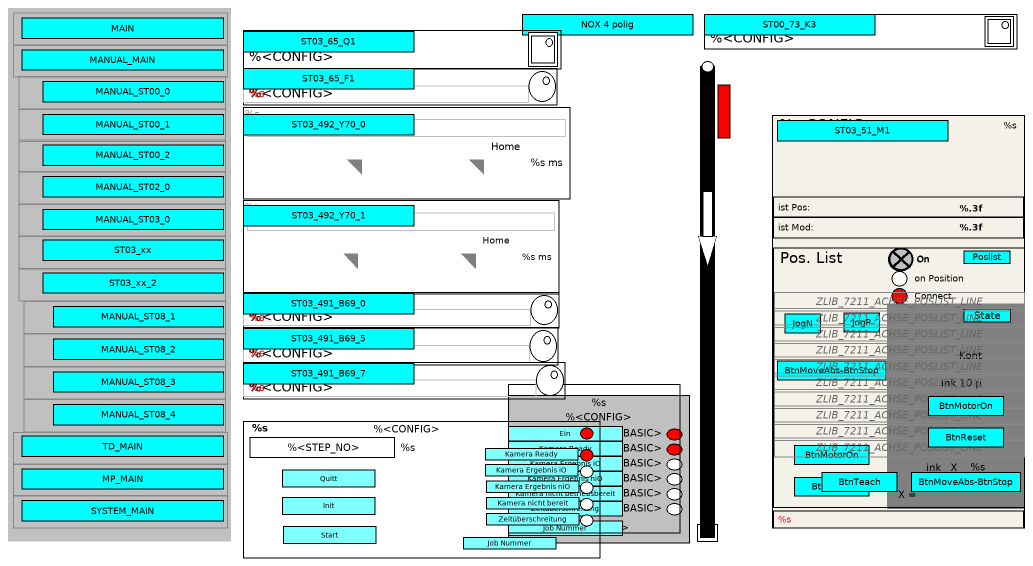
[picture p109: MANUAL_ST03_11 (HMI screen)]
embedded screen at (3,115)-(226,648): M0000_Manual
embedded screen at (238,214)-(565,306): ZLIB_VALVE_1_SENSORS
embedded screen at (238,307)-(554,401): ZLIB_VALVE_1_SENSORS
embedded screen at (238,399)-(554,435): VDIGIN
embedded screen at (238,434)-(553,472): VDIGIN
embedded screen at (767,222)-(1021,635): ZLIB_7211_Achse
embedded screen at (503,168)-(725,650): ZUFUEHRUNG_NOX_4POL
rectangle at (517,121)-(688,142): text "NOX 4 polig"; invisible if TRUE
rectangle at (238,312)-(409,333): text "ST03_492_Y70_1"; invisible if TRUE
rectangle at (238,221)-(409,242): text "ST03_492_Y70_0"; invisible if TRUE
rectangle at (238,400)-(409,421): text "ST03_491_B69_0"; invisible if TRUE
rectangle at (238,435)-(409,456): text "ST03_491_B69_5"; invisible if TRUE
rectangle at (772,227)-(943,248): text "ST03_51_M1"; invisible if TRUE
embedded screen at (238,137)-(556,176): VDIGOUT_SMAL
rectangle at (238,138)-(409,159): text "ST03_65_Q1"; invisible if TRUE
embedded screen at (238,175)-(552,212): VDIGIN
rectangle at (238,175)-(409,196): text "ST03_65_F1"; invisible if TRUE
embedded screen at (699,121)-(1012,156): VDIGOUT_SMAL
rectangle at (699,121)-(870,142): text "ST00_73_K3"; invisible if TRUE
embedded screen at (238,528)-(595,665): ZLIB_SENSOPART_4
embedded screen at (238,469)-(560,506): VDIGIN
rectangle at (238,470)-(409,491): text "ST03_491_B69_7"; invisible if TRUE
1 more shapes without text or variables
*)

(* Visualisation 01_ManualMode/ST03/MANUAL_ST03_12
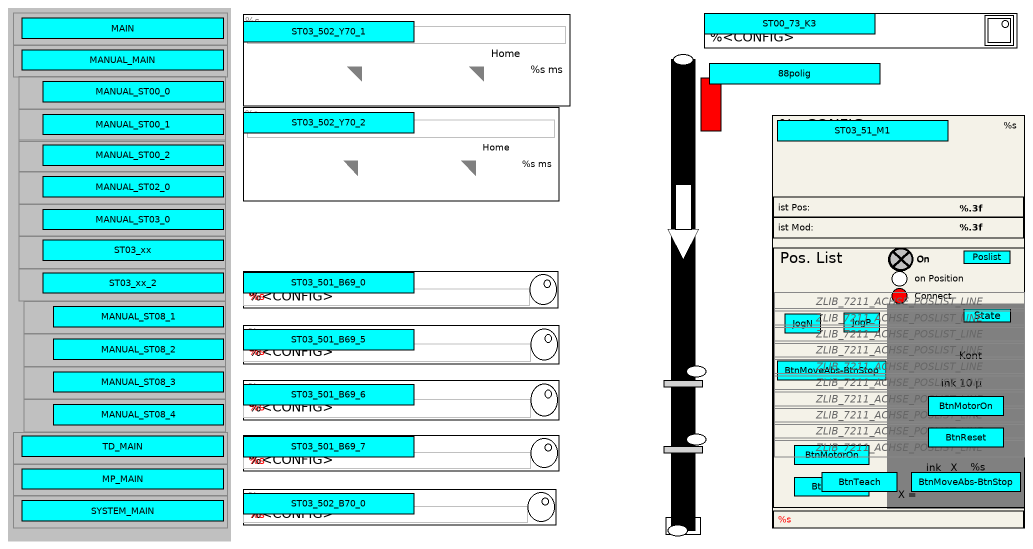
embedded screen at (3,115)-(226,648): M0000_Manual
embedded screen at (238,121)-(565,213): ZLIB_VALVE_1_SENSORS
embedded screen at (238,214)-(554,308): ZLIB_VALVE_1_SENSORS
embedded screen at (238,542)-(554,578): VDIGIN
embedded screen at (238,596)-(551,632): VDIGIN
embedded screen at (767,222)-(1021,635): ZLIB_7211_Achse
embedded screen at (646,161)-(716,643): ZUFUEHRUNG_88POL
rectangle at (704,170)-(875,191): text "88polig"; invisible if TRUE
rectangle at (238,219)-(409,240): text "ST03_502_Y70_2"; invisible if TRUE
rectangle at (238,128)-(409,149): text "ST03_502_Y70_1"; invisible if TRUE
rectangle at (238,543)-(409,564): text "ST03_501_B69_7"; invisible if TRUE
rectangle at (238,600)-(409,621): text "ST03_502_B70_0"; invisible if TRUE
rectangle at (772,227)-(943,248): text "ST03_51_M1"; invisible if TRUE
embedded screen at (238,487)-(554,527): VDIGIN
embedded screen at (238,378)-(553,415): VDIGIN
embedded screen at (238,432)-(554,471): VDIGIN
rectangle at (238,379)-(409,400): text "ST03_501_B69_0"; invisible if TRUE
rectangle at (238,436)-(409,457): text "ST03_501_B69_5"; invisible if TRUE
rectangle at (238,491)-(409,512): text "ST03_501_B69_6"; invisible if TRUE
embedded screen at (699,120)-(1012,155): VDIGOUT_SMAL
rectangle at (699,120)-(870,141): text "ST00_73_K3"; invisible if TRUE
*)

(* Visualisation 01_ManualMode/ST03/MANUAL_ST03_13
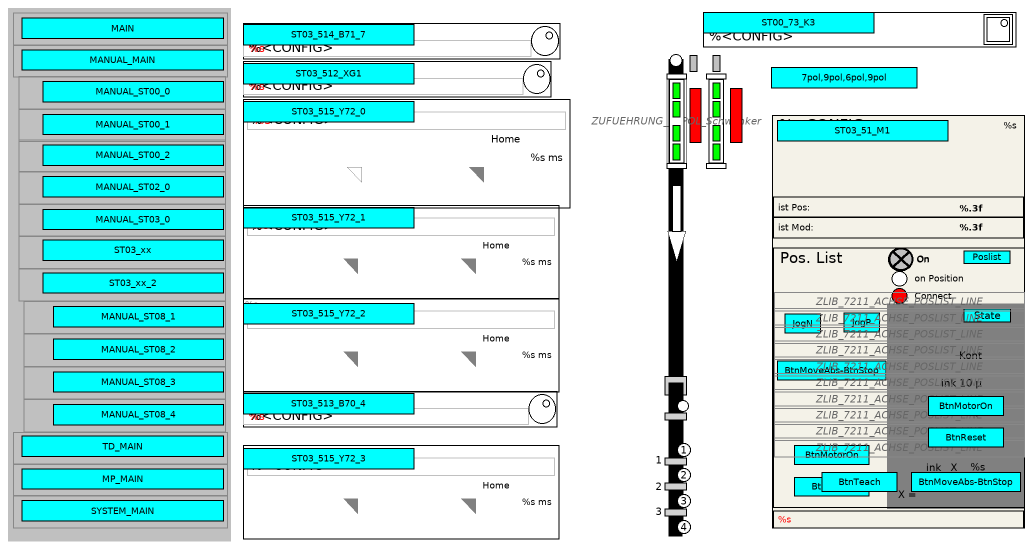
embedded screen at (3,115)-(226,648): M0000_Manual
embedded screen at (238,312)-(554,406): ZLIB_VALVE_1_SENSORS
embedded screen at (238,130)-(555,166): VDIGIN
embedded screen at (767,222)-(1021,635): ZLIB_7211_Achse
embedded screen at (646,161)-(737,643): ZUFUEHRUNG_7POL
rectangle at (766,174)-(912,195): text "7pol,9pol,6pol,9pol"; invisible if TRUE
rectangle at (238,314)-(409,335): text "ST03_515_Y72_1"; invisible if TRUE
rectangle at (238,131)-(409,152): text "ST03_514_B71_7"; invisible if TRUE
rectangle at (772,227)-(943,248): text "ST03_51_M1"; invisible if TRUE
embedded screen at (238,168)-(546,204): VDIGIN
rectangle at (238,170)-(409,191): text "ST03_512_XG1"; invisible if TRUE
embedded screen at (238,405)-(554,499): ZLIB_VALVE_1_SENSORS
embedded screen at (238,498)-(552,534): VDIGIN
rectangle at (238,410)-(409,431): text "ST03_515_Y72_2"; invisible if TRUE
rectangle at (238,500)-(409,521): text "ST03_513_B70_4"; invisible if TRUE
embedded screen at (238,552)-(554,646): ZLIB_VALVE_1_SENSORS
rectangle at (238,555)-(409,576): text "ST03_515_Y72_3"; invisible if TRUE
embedded screen at (238,206)-(565,315): ZLIB_VALVE_2_SENSORS
rectangle at (238,208)-(409,229): text "ST03_515_Y72_0"; invisible if TRUE
embedded screen at (698,119)-(1011,154): VDIGOUT_SMAL
rectangle at (698,119)-(869,140): text "ST00_73_K3"; invisible if TRUE
*)

(* Visualisation 01_ManualMode/ST03/MANUAL_ST03_13_2
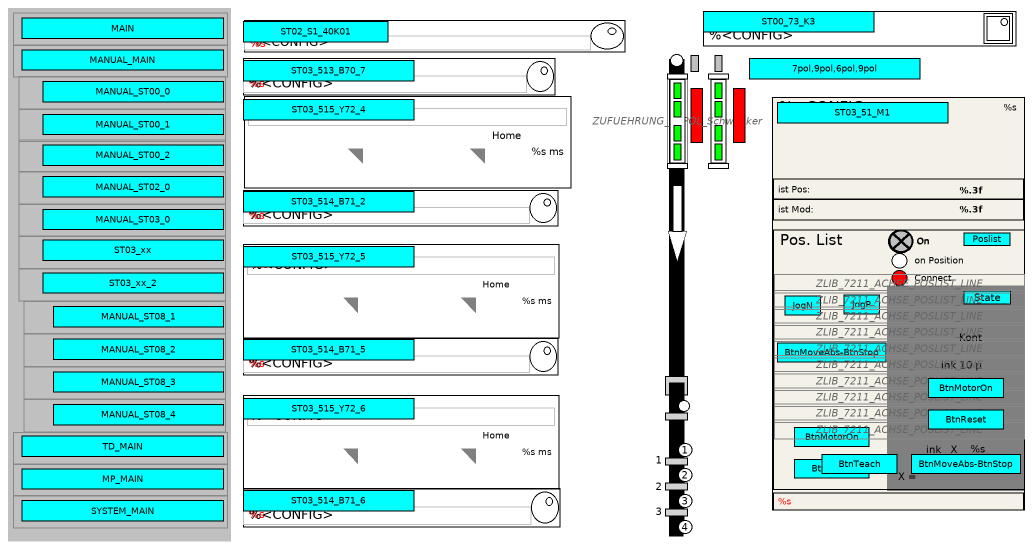
embedded screen at (3,115)-(226,648): M0000_Manual
embedded screen at (239,203)-(566,295): ZLIB_VALVE_1_SENSORS
embedded screen at (238,351)-(554,445): ZLIB_VALVE_1_SENSORS
embedded screen at (238,445)-(553,482): VDIGIN
embedded screen at (767,204)-(1021,617): ZLIB_7211_Achse
embedded screen at (646,161)-(740,643): ZUFUEHRUNG_7POL
rectangle at (744,165)-(915,186): text "7pol,9pol,6pol,9pol"; invisible if TRUE
rectangle at (238,353)-(409,374): text "ST03_515_Y72_5"; invisible if TRUE
rectangle at (238,206)-(409,227): text "ST03_515_Y72_4"; invisible if TRUE
rectangle at (238,446)-(409,467): text "ST03_514_B71_5"; invisible if TRUE
rectangle at (772,209)-(943,230): text "ST03_51_M1"; invisible if TRUE
embedded screen at (238,165)-(550,202): VDIGIN
rectangle at (238,167)-(409,188): text "ST03_513_B70_7"; invisible if TRUE
embedded screen at (238,502)-(554,596): ZLIB_VALVE_1_SENSORS
embedded screen at (238,595)-(555,634): VDIGIN
rectangle at (238,505)-(409,526): text "ST03_515_Y72_6"; invisible if TRUE
rectangle at (238,597)-(409,618): text "ST03_514_B71_6"; invisible if TRUE
embedded screen at (238,297)-(553,333): VDIGIN
rectangle at (238,298)-(409,319): text "ST03_514_B71_2"; invisible if TRUE
embedded screen at (239,127)-(620,159): VDIGIN
rectangle at (238,128)-(383,149): text "ST02_S1_40K01"; invisible if TRUE
embedded screen at (698,118)-(1011,153): VDIGOUT_SMAL
rectangle at (698,118)-(869,139): text "ST00_73_K3"; invisible if TRUE
*)

(* Visualisation 01_ManualMode/ST03/MANUAL_ST03_14
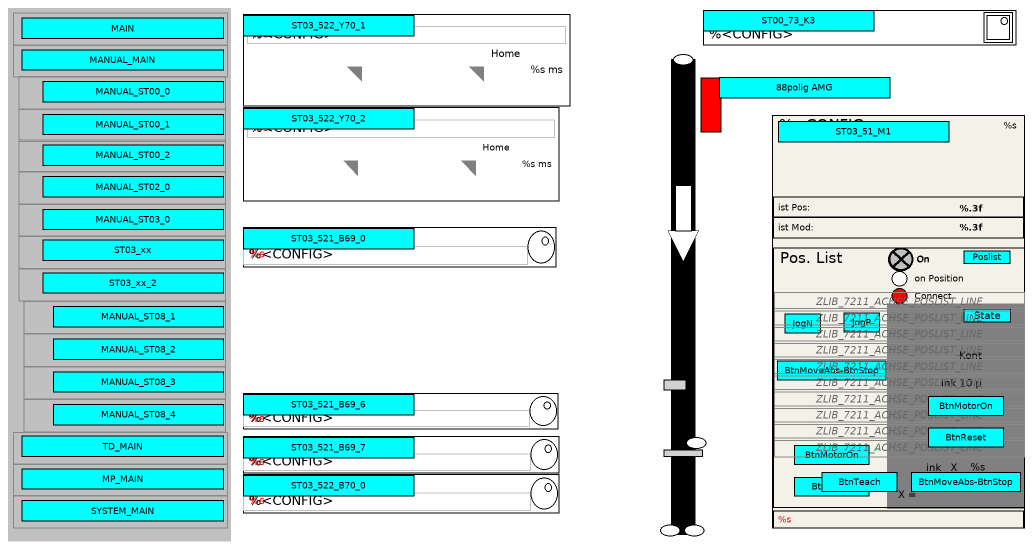
embedded screen at (3,115)-(226,648): M0000_Manual
embedded screen at (238,121)-(565,213): ZLIB_VALVE_1_SENSORS
embedded screen at (238,214)-(554,308): ZLIB_VALVE_1_SENSORS
embedded screen at (238,543)-(554,580): VDIGIN
embedded screen at (238,581)-(554,620): VDIGIN
embedded screen at (767,222)-(1021,635): ZLIB_7211_Achse
embedded screen at (646,161)-(716,643): ZUFUEHRUNG_88POL_AMG
rectangle at (714,184)-(885,205): text "88polig AMG"; invisible if TRUE
rectangle at (238,215)-(409,236): text "ST03_522_Y70_2"; invisible if TRUE
rectangle at (238,122)-(409,143): text "ST03_522_Y70_1"; invisible if TRUE
rectangle at (238,544)-(409,565): text "ST03_521_B69_7"; invisible if TRUE
rectangle at (238,582)-(409,603): text "ST03_522_B70_0"; invisible if TRUE
rectangle at (773,228)-(944,249): text "ST03_51_M1"; invisible if TRUE
embedded screen at (238,500)-(553,536): VDIGIN
embedded screen at (238,334)-(551,374): VDIGIN
rectangle at (238,335)-(409,356): text "ST03_521_B69_0"; invisible if TRUE
rectangle at (238,501)-(409,522): text "ST03_521_B69_6"; invisible if TRUE
embedded screen at (698,117)-(1011,152): VDIGOUT_SMAL
rectangle at (698,117)-(869,138): text "ST00_73_K3"; invisible if TRUE
*)

(* Visualisation 01_ManualMode/ST03/MANUAL_ST03_15
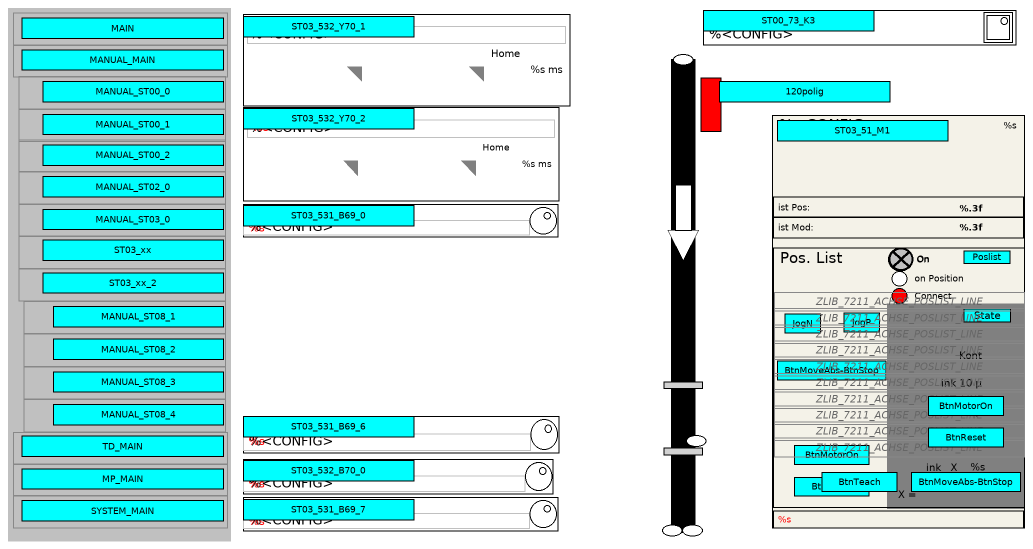
embedded screen at (3,115)-(226,648): M0000_Manual
embedded screen at (238,121)-(565,213): ZLIB_VALVE_1_SENSORS
embedded screen at (238,214)-(554,308): ZLIB_VALVE_1_SENSORS
embedded screen at (238,604)-(553,638): VDIGIN
embedded screen at (238,566)-(548,601): VDIGIN
embedded screen at (767,222)-(1021,635): ZLIB_7211_Achse
embedded screen at (646,161)-(716,643): ZUFUEHRUNG_120POL
rectangle at (714,188)-(885,209): text "120polig"; invisible if TRUE
rectangle at (238,215)-(409,236): text "ST03_532_Y70_2"; invisible if TRUE
rectangle at (238,123)-(409,144): text "ST03_532_Y70_1"; invisible if TRUE
rectangle at (238,606)-(409,627): text "ST03_531_B69_7"; invisible if TRUE
rectangle at (238,567)-(409,588): text "ST03_532_B70_0"; invisible if TRUE
rectangle at (772,227)-(943,248): text "ST03_51_M1"; invisible if TRUE
embedded screen at (238,523)-(554,560): VDIGIN
embedded screen at (238,311)-(553,344): VDIGIN
rectangle at (238,312)-(409,333): text "ST03_531_B69_0"; invisible if TRUE
rectangle at (238,523)-(409,544): text "ST03_531_B69_6"; invisible if TRUE
embedded screen at (698,117)-(1011,152): VDIGOUT_SMAL
rectangle at (698,117)-(869,138): text "ST00_73_K3"; invisible if TRUE
*)

(* Visualisation 01_ManualMode/ST03/MANUAL_ST03_16
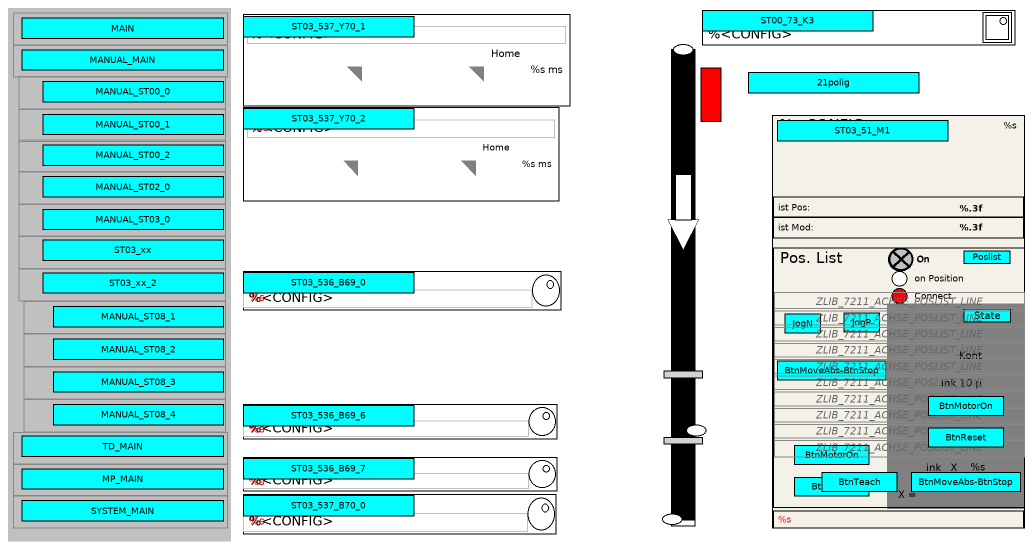
embedded screen at (3,115)-(226,648): M0000_Manual
embedded screen at (238,121)-(565,213): ZLIB_VALVE_1_SENSORS
embedded screen at (238,214)-(554,308): ZLIB_VALVE_1_SENSORS
embedded screen at (238,564)-(552,598): VDIGIN
embedded screen at (238,601)-(551,641): VDIGIN
embedded screen at (767,222)-(1021,635): ZLIB_7211_Achse
embedded screen at (646,151)-(716,633): ZUFUEHRUNG_21POL
rectangle at (743,179)-(914,200): text "21polig"; invisible if TRUE
rectangle at (238,215)-(409,236): text "ST03_537_Y70_2"; invisible if TRUE
rectangle at (238,123)-(409,144): text "ST03_537_Y70_1"; invisible if TRUE
rectangle at (238,565)-(409,586): text "ST03_536_B69_7"; invisible if TRUE
rectangle at (238,602)-(409,623): text "ST03_537_B70_0"; invisible if TRUE
rectangle at (772,227)-(943,248): text "ST03_51_M1"; invisible if TRUE
embedded screen at (238,511)-(552,546): VDIGIN
embedded screen at (238,378)-(556,417): VDIGIN
rectangle at (238,379)-(409,400): text "ST03_536_B69_0"; invisible if TRUE
rectangle at (238,512)-(409,533): text "ST03_536_B69_6"; invisible if TRUE
embedded screen at (697,117)-(1010,152): VDIGOUT_SMAL
rectangle at (697,117)-(868,138): text "ST00_73_K3"; invisible if TRUE
*)

(* Visualisation 01_ManualMode/ST03/MANUAL_ST03_17
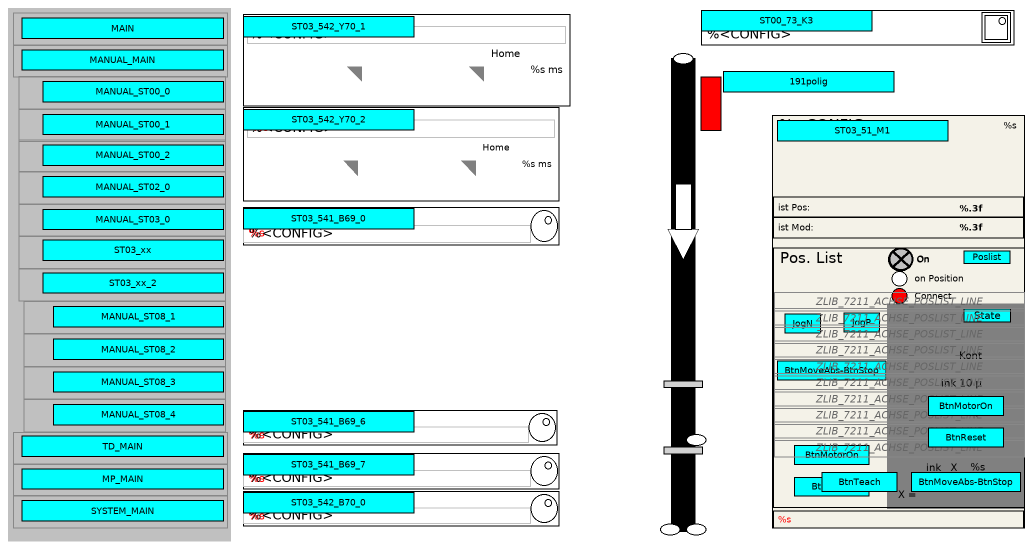
embedded screen at (3,115)-(226,648): M0000_Manual
embedded screen at (238,121)-(565,213): ZLIB_VALVE_1_SENSORS
embedded screen at (238,214)-(554,308): ZLIB_VALVE_1_SENSORS
embedded screen at (238,560)-(554,596): VDIGIN
embedded screen at (238,598)-(554,633): VDIGIN
embedded screen at (767,222)-(1021,635): ZLIB_7211_Achse
embedded screen at (646,160)-(716,642): ZUFUEHRUNG_191POL
rectangle at (718,178)-(889,199): text "191polig"; invisible if TRUE
rectangle at (238,216)-(409,237): text "ST03_542_Y70_2"; invisible if TRUE
rectangle at (238,123)-(409,144): text "ST03_542_Y70_1"; invisible if TRUE
rectangle at (238,561)-(409,582): text "ST03_541_B69_7"; invisible if TRUE
rectangle at (238,599)-(409,620): text "ST03_542_B70_0"; invisible if TRUE
rectangle at (772,227)-(943,248): text "ST03_51_M1"; invisible if TRUE
embedded screen at (238,517)-(552,552): VDIGIN
embedded screen at (238,314)-(554,352): VDIGIN
rectangle at (238,315)-(409,336): text "ST03_541_B69_0"; invisible if TRUE
rectangle at (238,518)-(409,539): text "ST03_541_B69_6"; invisible if TRUE
embedded screen at (696,117)-(1009,152): VDIGOUT_SMAL
rectangle at (696,117)-(867,138): text "ST00_73_K3"; invisible if TRUE
*)

(* Visualisation 01_ManualMode/ST03/MANUAL_ST03_18
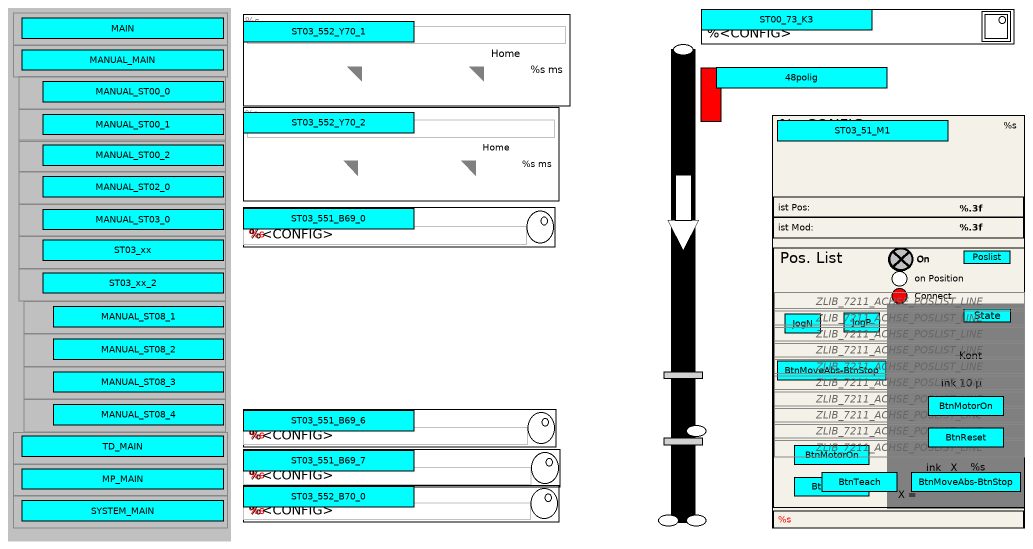
embedded screen at (3,115)-(226,648): M0000_Manual
embedded screen at (238,121)-(565,213): ZLIB_VALVE_1_SENSORS
embedded screen at (238,214)-(554,308): ZLIB_VALVE_1_SENSORS
embedded screen at (238,556)-(555,594): VDIGIN
embedded screen at (238,592)-(554,629): VDIGIN
embedded screen at (767,222)-(1021,635): ZLIB_7211_Achse
embedded screen at (646,151)-(716,633): ZUFUEHRUNG_48POL
rectangle at (711,174)-(882,195): text "48polig"; invisible if TRUE
rectangle at (238,219)-(409,240): text "ST03_552_Y70_2"; invisible if TRUE
rectangle at (238,128)-(409,149): text "ST03_552_Y70_1"; invisible if TRUE
rectangle at (238,557)-(409,578): text "ST03_551_B69_7"; invisible if TRUE
rectangle at (238,593)-(409,614): text "ST03_552_B70_0"; invisible if TRUE
rectangle at (772,227)-(943,248): text "ST03_51_M1"; invisible if TRUE
embedded screen at (238,516)-(551,554): VDIGIN
embedded screen at (238,314)-(550,354): VDIGIN
rectangle at (238,315)-(409,336): text "ST03_551_B69_0"; invisible if TRUE
rectangle at (238,517)-(409,538): text "ST03_551_B69_6"; invisible if TRUE
embedded screen at (696,116)-(1009,151): VDIGOUT_SMAL
rectangle at (696,116)-(867,137): text "ST00_73_K3"; invisible if TRUE
*)

(* Visualisation 01_ManualMode/ST03/MANUAL_ST03_19
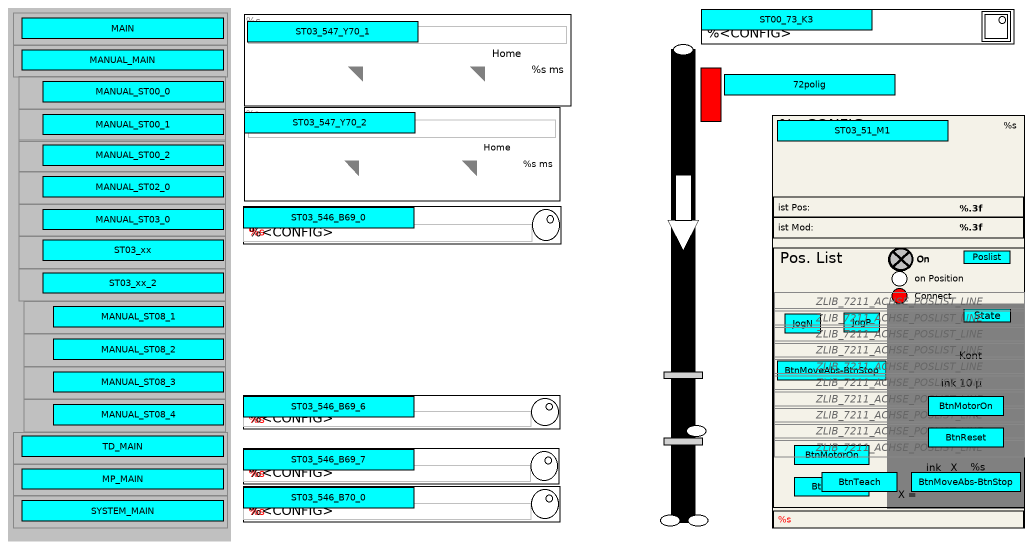
embedded screen at (3,115)-(226,648): M0000_Manual
embedded screen at (239,121)-(566,213): ZLIB_VALVE_1_SENSORS
embedded screen at (239,214)-(555,308): ZLIB_VALVE_1_SENSORS
embedded screen at (238,555)-(554,591): VDIGIN
embedded screen at (238,593)-(555,629): VDIGIN
embedded screen at (767,222)-(1021,635): ZLIB_7211_Achse
embedded screen at (646,151)-(716,633): ZUFUEHRUNG_72POL
rectangle at (719,181)-(890,202): text "72polig"; invisible if TRUE
rectangle at (239,219)-(410,240): text "ST03_547_Y70_2"; invisible if TRUE
rectangle at (242,128)-(413,149): text "ST03_547_Y70_1"; invisible if TRUE
rectangle at (238,556)-(409,577): text "ST03_546_B69_7"; invisible if TRUE
rectangle at (238,594)-(409,615): text "ST03_546_B70_0"; invisible if TRUE
rectangle at (772,227)-(943,248): text "ST03_51_M1"; invisible if TRUE
embedded screen at (238,502)-(555,536): VDIGIN
embedded screen at (238,313)-(556,351): VDIGIN
rectangle at (238,314)-(409,335): text "ST03_546_B69_0"; invisible if TRUE
rectangle at (238,503)-(409,524): text "ST03_546_B69_6"; invisible if TRUE
embedded screen at (696,116)-(1009,151): VDIGOUT_SMAL
rectangle at (696,116)-(867,137): text "ST00_73_K3"; invisible if TRUE
*)

(* Visualisation 01_ManualMode/ST03/MANUAL_ST03_2
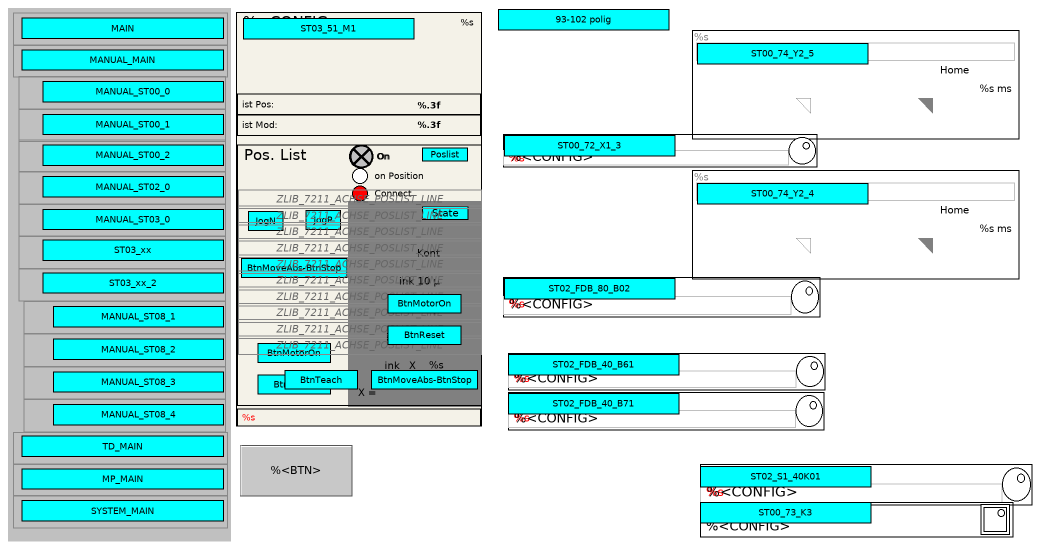
embedded screen at (3,115)-(226,648): M0000_Manual
embedded screen at (687,277)-(1014,386): ZLIB_VALVE_2_SENSORS
embedded screen at (687,137)-(1014,246): ZLIB_VALVE_2_SENSORS
embedded screen at (231,119)-(478,533): ZLIB_7211_Achse
embedded screen at (695,571)-(1027,612): VDIGIN
embedded screen at (498,241)-(812,274): VDIGIN
embedded screen at (498,384)-(815,424): VDIGIN
button at (235,552)-(347,603): text "%<BTN>"; shows 'TaktBand'; invisible if gTypeCode<>4991 AND gTypeCode <>312; taps ST03_Band.b_MoveRel
embedded screen at (503,460)-(820,497): VDIGIN
embedded screen at (503,499)-(819,537): VDIGIN
rectangle at (493,116)-(664,137): text "93-102 polig"; invisible if TRUE
rectangle at (238,125)-(409,146): text "ST03_51_M1"; invisible if TRUE
rectangle at (695,573)-(866,594): text "ST02_S1_40K01"; invisible if TRUE
rectangle at (503,461)-(674,482): text "ST02_FDB_40_B61"; invisible if TRUE
rectangle at (503,500)-(674,521): text "ST02_FDB_40_B71"; invisible if TRUE
rectangle at (499,385)-(670,406): text "ST02_FDB_80_B02"; invisible if TRUE
rectangle at (499,242)-(670,263): text "ST00_72_X1_3"; invisible if TRUE
rectangle at (692,150)-(863,171): text "ST00_74_Y2_5"; invisible if TRUE
rectangle at (692,290)-(863,311): text "ST00_74_Y2_4"; invisible if TRUE
embedded screen at (695,609)-(1008,644): VDIGOUT_SMAL
rectangle at (695,609)-(866,630): text "ST00_73_K3"; invisible if TRUE
*)

(* Visualisation 01_ManualMode/ST03/MANUAL_ST03_20
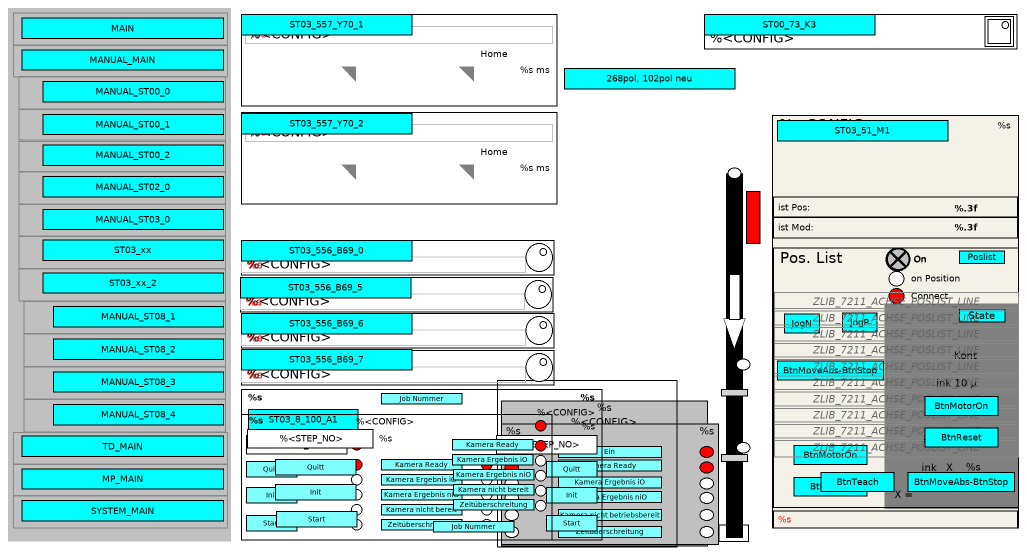
embedded screen at (3,115)-(226,648): M0000_Manual
embedded screen at (699,121)-(1012,156): VDIGOUT_SMAL
embedded screen at (236,121)-(552,213): ZLIB_VALVE_1_SENSORS
embedded screen at (236,219)-(552,311): ZLIB_VALVE_1_SENSORS
embedded screen at (767,222)-(1015,635): ZLIB_7211_Achse
embedded screen at (496,176)-(755,653): ZUFUEHRUNG_268POL_102POL_NEU
rectangle at (559,175)-(730,196): text "268pol, 102pol neu"; invisible if TRUE
rectangle at (236,220)-(407,241): text "ST03_557_Y70_2"; invisible if TRUE
rectangle at (236,121)-(407,142): text "ST03_557_Y70_1"; invisible if TRUE
rectangle at (699,121)-(870,142): text "ST00_73_K3"; invisible if TRUE
rectangle at (772,227)-(943,248): text "ST03_51_M1"; invisible if TRUE
embedded screen at (236,420)-(549,455): VDIGIN
embedded screen at (236,347)-(549,382): VDIGIN
rectangle at (236,347)-(407,368): text "ST03_556_B69_0"; invisible if TRUE
rectangle at (236,420)-(407,441): text "ST03_556_B69_6"; invisible if TRUE
embedded screen at (236,496)-(597,647): ZLIB_SENSOPART_4_2
embedded screen at (235,384)-(548,419): VDIGIN
rectangle at (235,384)-(406,405): text "ST03_556_B69_5"; invisible if TRUE
rectangle at (243,516)-(353,537): text "ST03_8_100_A1"; invisible if TRUE
embedded screen at (236,457)-(549,492): VDIGIN
rectangle at (236,456)-(407,477): text "ST03_556_B69_7"; invisible if TRUE
embedded screen at (236,521)-(547,647): ZLIB_SENSOPART_4
1 more shapes without text or variables
*)

(* Visualisation 01_ManualMode/ST03/MANUAL_ST03_20_2
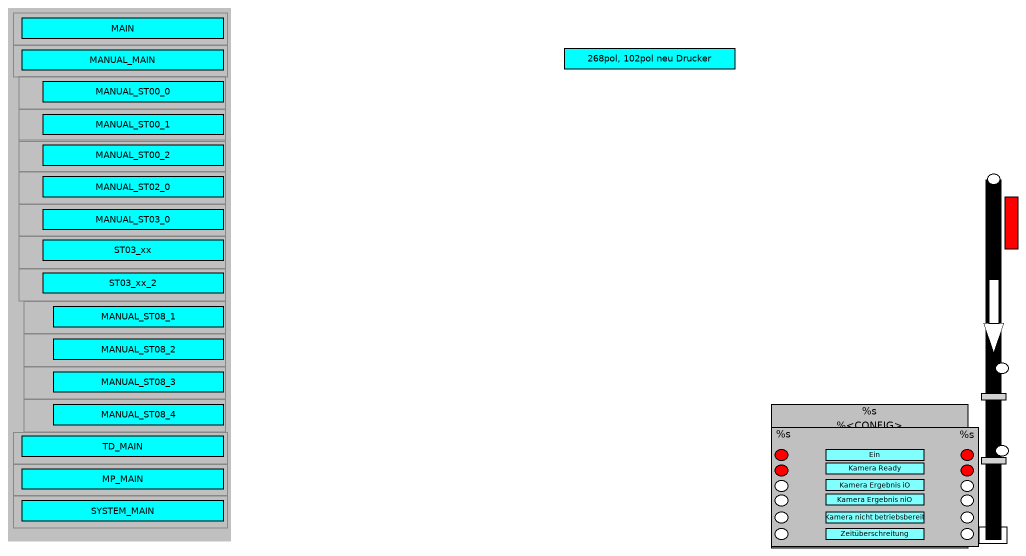
embedded screen at (766,183)-(1013,655): ZUFUEHRUNG_268POL_102POL_NEU
embedded screen at (3,115)-(226,648): M0000_Manual
rectangle at (559,155)-(730,176): text "268pol, 102pol neu Drucker"; invisible if TRUE
*)

(* Visualisation 01_ManualMode/ST03/MANUAL_ST03_21
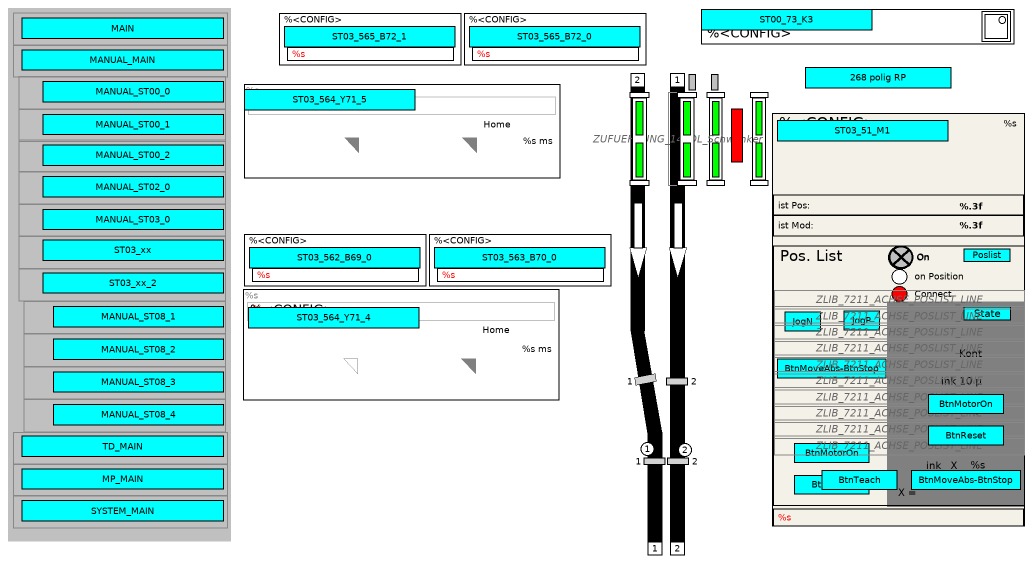
embedded screen at (3,115)-(226,648): M0000_Manual
embedded screen at (239,191)-(555,285): ZLIB_VALVE_1_SENSORS
embedded screen at (459,120)-(641,172): ZLIB_DIG_IN
embedded screen at (767,220)-(1021,633): ZLIB_7211_Achse
embedded screen at (590,180)-(763,662): ZUFUEHRUNG_268POL_RP
rectangle at (800,174)-(946,195): text "268 polig RP"; invisible if TRUE
rectangle at (239,196)-(410,217): text "ST03_564_Y71_5"; invisible if TRUE
rectangle at (464,133)-(635,154): text "ST03_565_B72_0"; invisible if TRUE
rectangle at (772,227)-(943,248): text "ST03_51_M1"; invisible if TRUE
embedded screen at (274,120)-(456,172): ZLIB_DIG_IN
rectangle at (279,133)-(450,154): text "ST03_565_B72_1"; invisible if TRUE
embedded screen at (239,341)-(421,393): ZLIB_DIG_IN
rectangle at (244,354)-(415,375): text "ST03_562_B69_0"; invisible if TRUE
embedded screen at (238,396)-(554,507): ZLIB_VALVE_2_SENSORS
rectangle at (243,414)-(414,435): text "ST03_564_Y71_4"; invisible if TRUE
embedded screen at (424,341)-(606,393): ZLIB_DIG_IN
rectangle at (429,354)-(600,375): text "ST03_563_B70_0"; invisible if TRUE
embedded screen at (696,116)-(1009,151): VDIGOUT_SMAL
rectangle at (696,116)-(867,137): text "ST00_73_K3"; invisible if TRUE
*)

(* Visualisation 01_ManualMode/ST03/MANUAL_ST03_21_2
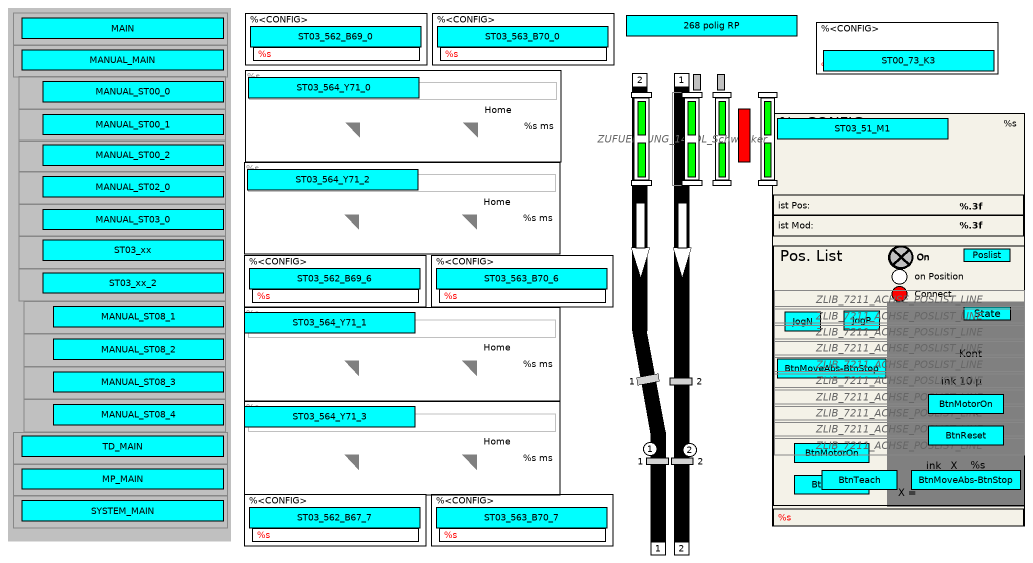
embedded screen at (3,115)-(226,648): M0000_Manual
embedded screen at (811,129)-(993,181): ZLIB_DIGOUT
embedded screen at (239,269)-(555,361): ZLIB_VALVE_1_SENSORS
embedded screen at (239,414)-(555,508): ZLIB_VALVE_1_SENSORS
embedded screen at (426,601)-(608,653): ZLIB_DIG_IN
embedded screen at (767,220)-(1021,633): ZLIB_7211_Achse
embedded screen at (590,180)-(772,662): ZUFUEHRUNG_268POL_RP
rectangle at (621,122)-(792,143): text "268 polig RP"; invisible if TRUE
rectangle at (239,419)-(410,440): text "ST03_564_Y71_1"; invisible if TRUE
rectangle at (242,276)-(413,297): text "ST03_564_Y71_2"; invisible if TRUE
rectangle at (431,614)-(602,635): text "ST03_563_B70_7"; invisible if TRUE
rectangle at (818,157)-(989,178): text "ST00_73_K3"; invisible if TRUE
rectangle at (772,225)-(943,246): text "ST03_51_M1"; invisible if TRUE
embedded screen at (426,362)-(608,414): ZLIB_DIG_IN
rectangle at (431,375)-(602,396): text "ST03_563_B70_6"; invisible if TRUE
embedded screen at (239,508)-(555,602): ZLIB_VALVE_1_SENSORS
embedded screen at (239,601)-(421,653): ZLIB_DIG_IN
rectangle at (239,513)-(410,534): text "ST03_564_Y71_3"; invisible if TRUE
rectangle at (244,614)-(415,635): text "ST03_562_B67_7"; invisible if TRUE
embedded screen at (239,362)-(421,414): ZLIB_DIG_IN
rectangle at (244,375)-(415,396): text "ST03_562_B69_6"; invisible if TRUE
embedded screen at (240,177)-(556,269): ZLIB_VALVE_1_SENSORS
rectangle at (243,184)-(414,205): text "ST03_564_Y71_0"; invisible if TRUE
embedded screen at (427,120)-(609,172): ZLIB_DIG_IN
rectangle at (432,133)-(603,154): text "ST03_563_B70_0"; invisible if TRUE
embedded screen at (240,120)-(422,172): ZLIB_DIG_IN
rectangle at (245,133)-(416,154): text "ST03_562_B69_0"; invisible if TRUE
*)

(* Visualisation 01_ManualMode/ST03/MANUAL_ST03_22
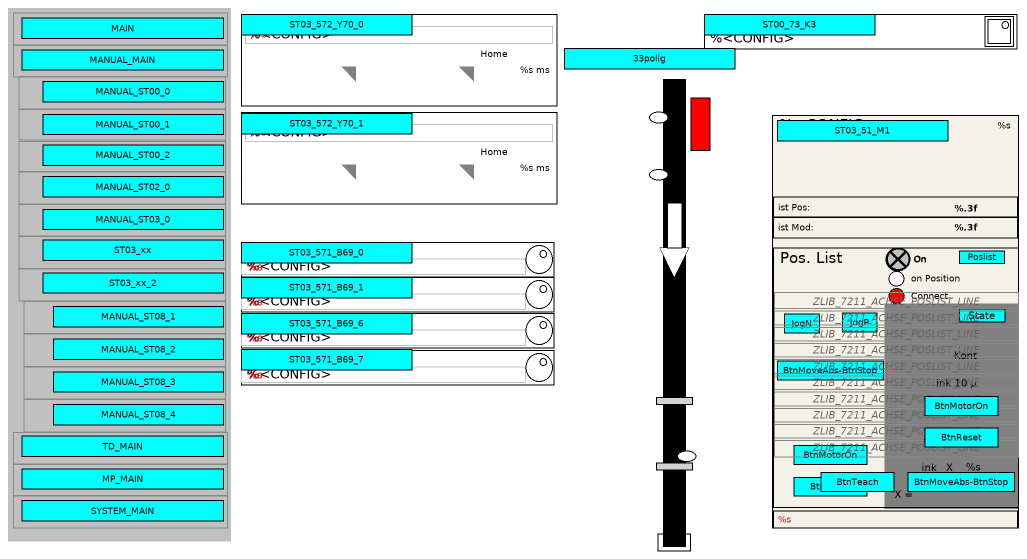
embedded screen at (3,115)-(226,648): M0000_Manual
embedded screen at (699,121)-(1012,156): VDIGOUT_SMAL
embedded screen at (236,121)-(552,213): ZLIB_VALVE_1_SENSORS
embedded screen at (236,219)-(552,311): ZLIB_VALVE_1_SENSORS
embedded screen at (236,457)-(549,492): VDIGIN
embedded screen at (767,222)-(1015,635): ZLIB_7211_Achse
embedded screen at (639,181)-(705,658): ZUFUEHRUNG_33POL
rectangle at (559,155)-(730,176): text "33polig"; invisible if TRUE
rectangle at (236,220)-(407,241): text "ST03_572_Y70_1"; invisible if TRUE
rectangle at (236,121)-(407,142): text "ST03_572_Y70_0"; invisible if TRUE
rectangle at (236,456)-(407,477): text "ST03_571_B69_7"; invisible if TRUE
rectangle at (699,121)-(870,142): text "ST00_73_K3"; invisible if TRUE
rectangle at (772,227)-(943,248): text "ST03_51_M1"; invisible if TRUE
embedded screen at (236,420)-(549,455): VDIGIN
embedded screen at (236,384)-(549,419): VDIGIN
rectangle at (236,384)-(407,405): text "ST03_571_B69_1"; invisible if TRUE
rectangle at (236,420)-(407,441): text "ST03_571_B69_6"; invisible if TRUE
embedded screen at (236,349)-(549,384): VDIGIN
rectangle at (236,349)-(407,370): text "ST03_571_B69_0"; invisible if TRUE
*)

(* Visualisation 01_ManualMode/ST03/MANUAL_ST03_23
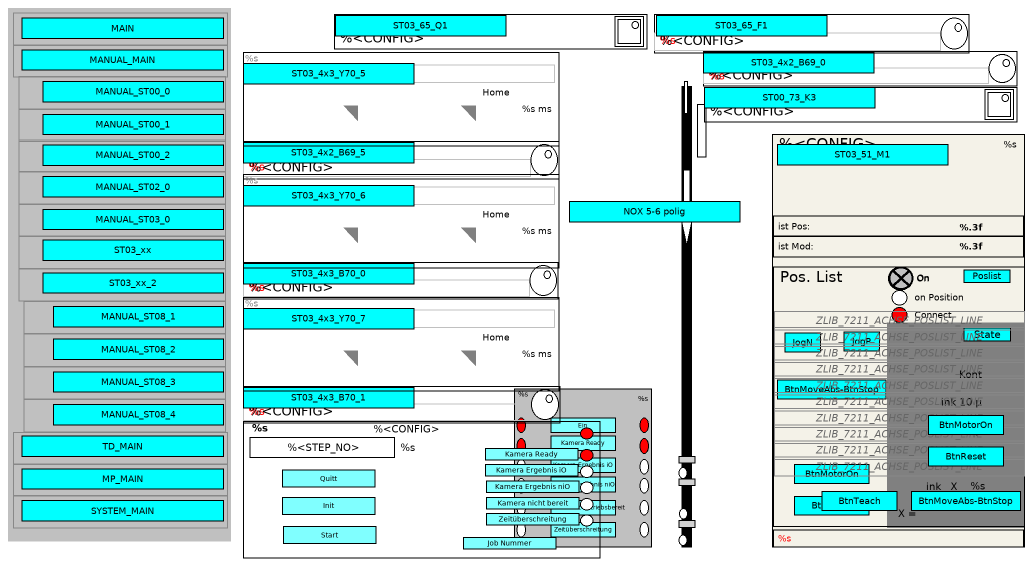
embedded screen at (3,115)-(226,648): M0000_Manual
embedded screen at (460,188)-(701,654): ZUFUEHRUNG_NOX_5_6POL
embedded screen at (238,493)-(555,530): VDIGIN
embedded screen at (698,158)-(1012,193): VDIGIN
embedded screen at (238,248)-(554,286): VDIGIN
embedded screen at (238,369)-(553,406): VDIGIN
embedded screen at (767,241)-(1021,654): ZLIB_7211_Achse
rectangle at (564,308)-(735,329): text "NOX 5-6 polig"; invisible if TRUE
rectangle at (698,159)-(869,180): text "ST03_4x2_B69_0"; invisible if TRUE
rectangle at (238,249)-(409,270): text "ST03_4x2_B69_5"; invisible if TRUE
rectangle at (238,494)-(409,515): text "ST03_4x3_B70_1"; invisible if TRUE
rectangle at (238,370)-(409,391): text "ST03_4x3_B70_0"; invisible if TRUE
rectangle at (772,251)-(943,272): text "ST03_51_M1"; invisible if TRUE
embedded screen at (238,159)-(554,253): ZLIB_VALVE_1_SENSORS
rectangle at (238,170)-(409,191): text "ST03_4x3_Y70_5"; invisible if TRUE
embedded screen at (238,281)-(554,375): ZLIB_VALVE_1_SENSORS
rectangle at (238,292)-(409,313): text "ST03_4x3_Y70_6"; invisible if TRUE
embedded screen at (238,404)-(554,498): ZLIB_VALVE_1_SENSORS
rectangle at (238,415)-(409,436): text "ST03_4x3_Y70_7"; invisible if TRUE
embedded screen at (329,121)-(642,156): VDIGOUT_SMAL
rectangle at (330,122)-(501,143): text "ST03_65_Q1"; invisible if TRUE
embedded screen at (649,121)-(964,160): VDIGIN
rectangle at (651,122)-(822,143): text "ST03_65_F1"; invisible if TRUE
embedded screen at (699,194)-(1012,229): VDIGOUT_SMAL
rectangle at (699,194)-(870,215): text "ST00_73_K3"; invisible if TRUE
embedded screen at (238,528)-(595,665): ZLIB_SENSOPART_4
*)

(* Visualisation 01_ManualMode/ST03/MANUAL_ST03_3
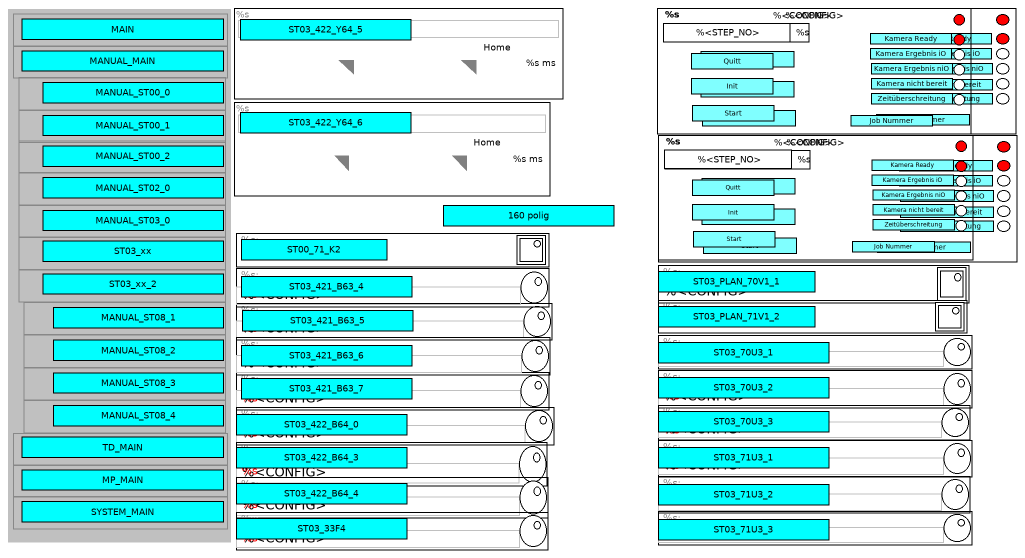
embedded screen at (3,115)-(226,648): M0000_MANUAL
embedded screen at (653,371)-(964,409): VDIGOUT_SMAL
embedded screen at (229,114)-(558,205): ZLIB_VALVE_1_SENSORS
embedded screen at (229,208)-(545,302): ZLIB_VALVE_1_SENSORS
embedded screen at (231,478)-(544,516): VDIGIN
embedded screen at (231,513)-(549,551): VDIGIN
embedded screen at (231,409)-(547,446): VDIGIN
embedded screen at (231,443)-(545,481): VDIGIN
embedded screen at (231,374)-(544,413): VDIGIN
embedded screen at (231,548)-(542,592): VDIGIN
embedded screen at (652,114)-(1011,240): ZLIB_SENSOPART
embedded screen at (653,241)-(1012,368): ZLIB_SENSOPART
embedded screen at (231,583)-(543,624): VDIGIN
embedded screen at (653,406)-(962,439): VDIGOUT_SMAL
embedded screen at (231,618)-(543,656): VDIGIN
embedded screen at (653,546)-(967,583): VDIGIN
embedded screen at (653,476)-(967,514): VDIGIN
embedded screen at (653,511)-(965,546): VDIGIN
embedded screen at (653,441)-(967,475): VDIGIN
embedded screen at (653,582)-(965,619): VDIGIN
embedded screen at (653,617)-(967,651): VDIGIN
embedded screen at (652,114)-(966,240): ZLIB_SENSOPART_4
embedded screen at (653,241)-(968,366): ZLIB_SENSOPART_4
rectangle at (438,311)-(609,332): text "160 polig"; invisible if TRUE
rectangle at (235,125)-(406,146): text "ST03_422_Y64_5"; invisible if TRUE
rectangle at (235,218)-(406,239): text "ST03_422_Y64_6"; invisible if TRUE
rectangle at (236,382)-(407,403): text "ST03_421_B63_4"; invisible if TRUE
rectangle at (231,520)-(402,541): text "ST03_422_B64_0"; invisible if TRUE
rectangle at (231,553)-(402,574): text "ST03_422_B64_3"; invisible if TRUE
rectangle at (237,416)-(408,437): text "ST03_421_B63_5"; invisible if TRUE
rectangle at (236,451)-(407,472): text "ST03_421_B63_6"; invisible if TRUE
rectangle at (231,589)-(402,610): text "ST03_422_B64_4"; invisible if TRUE
rectangle at (231,624)-(402,645): text "ST03_33F4"; invisible if TRUE
rectangle at (236,484)-(407,505): text "ST03_421_B63_7"; invisible if TRUE
rectangle at (653,448)-(824,469): text "ST03_70U3_1"; invisible if TRUE
rectangle at (653,483)-(824,504): text "ST03_70U3_2"; invisible if TRUE
rectangle at (653,517)-(824,538): text "ST03_70U3_3"; invisible if TRUE
rectangle at (653,553)-(824,574): text "ST03_71U3_1"; invisible if TRUE
rectangle at (653,590)-(824,611): text "ST03_71U3_2"; invisible if TRUE
rectangle at (653,625)-(824,646): text "ST03_71U3_3"; invisible if TRUE
rectangle at (653,377)-(810,398): text "ST03_PLAN_70V1_1"; invisible if TRUE
rectangle at (653,412)-(810,433): text "ST03_PLAN_71V1_2"; invisible if TRUE
embedded screen at (231,339)-(544,373): VDIGOUT_SMAL
rectangle at (236,345)-(382,366): text "ST00_71_K2"; invisible if TRUE
*)

(* Visualisation 01_ManualMode/ST03/MANUAL_ST03_3_2
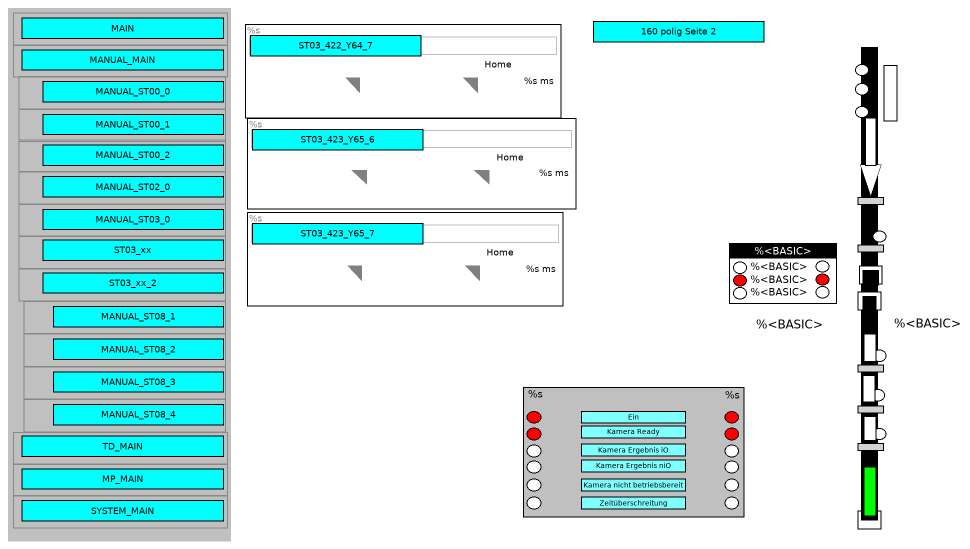
embedded screen at (3,115)-(226,648): M0000_MANUAL
embedded screen at (242,225)-(571,316): ZLIB_VALVE_1_SENSORS
embedded screen at (242,319)-(558,413): ZLIB_VALVE_1_SENSORS
embedded screen at (240,131)-(556,225): ZLIB_VALVE_1_SENSORS
rectangle at (588,128)-(759,149): text "160 polig Seite 2"; invisible if TRUE
embedded screen at (518,154)-(980,636): ZUFUEHRUNG_160POL
rectangle at (245,142)-(416,163): text "ST03_422_Y64_7"; invisible if TRUE
rectangle at (247,236)-(418,257): text "ST03_423_Y65_6"; invisible if TRUE
rectangle at (247,330)-(418,351): text "ST03_423_Y65_7"; invisible if TRUE
*)

(* Visualisation 01_ManualMode/ST03/MANUAL_ST03_4
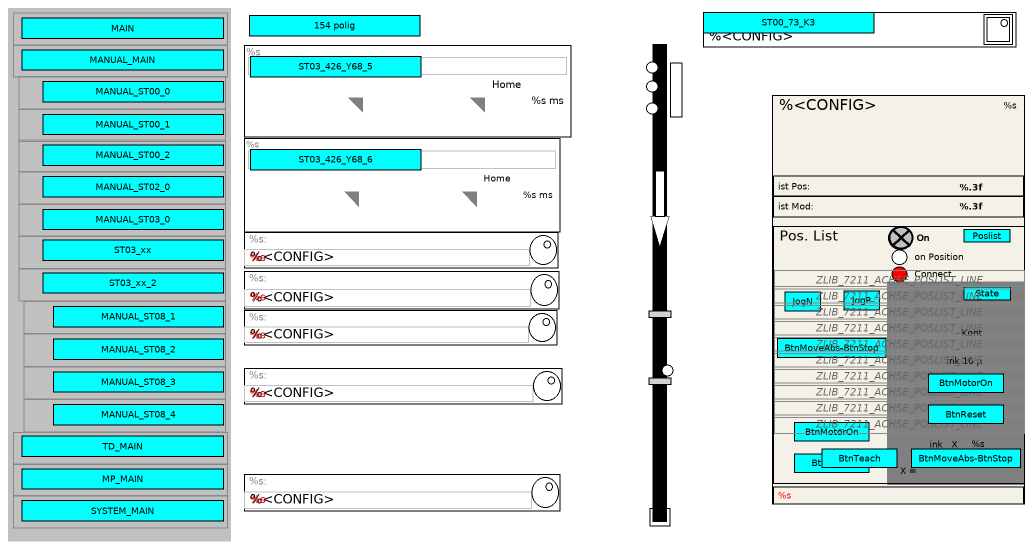
embedded screen at (3,115)-(226,648): M0000_Manual
embedded screen at (239,152)-(566,244): ZLIB_VALVE_1_SENSORS
embedded screen at (239,245)-(555,339): ZLIB_VALVE_1_SENSORS
embedded screen at (239,417)-(552,452): VDIGIN
embedded screen at (239,339)-(553,375): VDIGIN
embedded screen at (239,378)-(554,416): VDIGIN
embedded screen at (239,581)-(555,618): VDIGIN
embedded screen at (239,475)-(557,511): VDIGIN
embedded screen at (636,151)-(677,633): ZUFUEHRUNG_154POL
embedded screen at (767,202)-(1021,611): ZLIB_7211_Achse
rectangle at (244,122)-(415,143): text "154 polig"; invisible if TRUE
rectangle at (245,163)-(416,184): text "ST03_426_Y68_5"; invisible if TRUE
rectangle at (245,256)-(416,277): text "ST03_426_Y68_6"; invisible if TRUE
embedded screen at (698,119)-(1011,154): VDIGOUT_SMAL
rectangle at (698,119)-(869,140): text "ST00_73_K3"; invisible if TRUE
*)

(* Visualisation 01_ManualMode/ST03/MANUAL_ST03_5
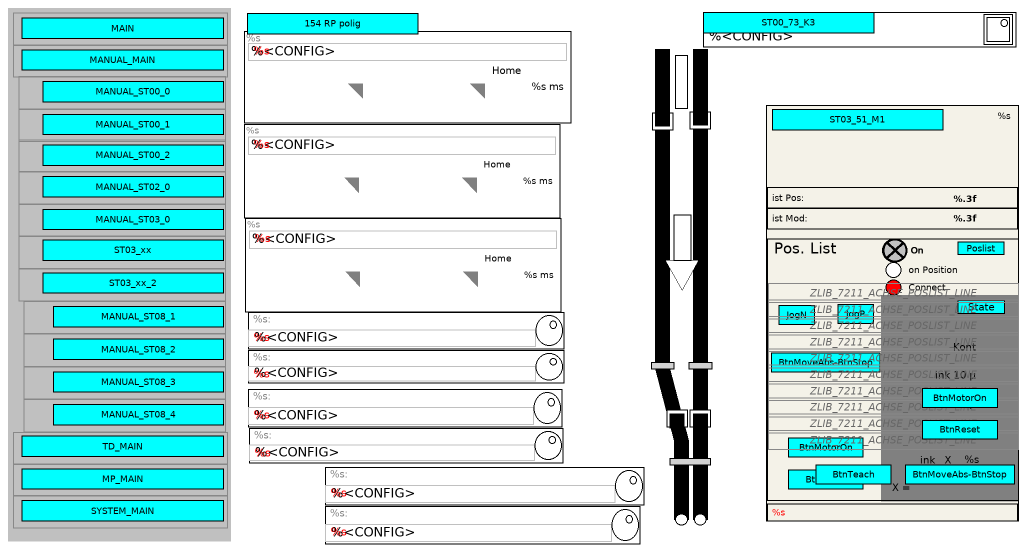
embedded screen at (3,115)-(226,648): M0000_Manual
embedded screen at (239,138)-(566,230): ZLIB_VALVE_1_SENSORS
embedded screen at (239,231)-(555,325): ZLIB_VALVE_1_SENSORS
embedded screen at (244,535)-(558,570): VDIGIN
embedded screen at (320,574)-(639,612): VDIGIN
embedded screen at (243,457)-(559,490): VDIGIN
embedded screen at (243,496)-(557,534): VDIGIN
embedded screen at (243,419)-(559,456): VDIGIN
embedded screen at (320,613)-(635,651): VDIGIN
embedded screen at (240,325)-(556,419): ZLIB_VALVE_1_SENSORS
embedded screen at (646,156)-(707,632): ZUFUEHRUNG_154RP
embedded screen at (761,212)-(1015,628): ZLIB_7211_Achse
rectangle at (242,120)-(413,141): text "154 RP polig"; invisible if TRUE
rectangle at (767,216)-(938,237): text "ST03_51_M1"; invisible if TRUE
embedded screen at (698,119)-(1011,154): VDIGOUT_SMAL
rectangle at (698,119)-(869,140): text "ST00_73_K3"; invisible if TRUE
*)

(* Visualisation 01_ManualMode/ST03/MANUAL_ST03_6
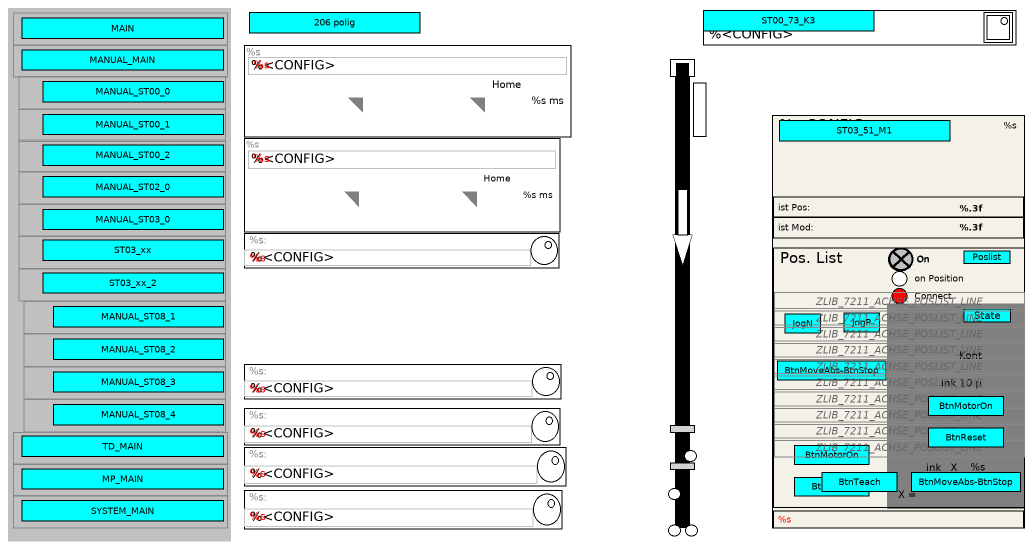
embedded screen at (3,115)-(226,648): M0000_Manual
embedded screen at (239,152)-(566,244): ZLIB_VALVE_1_SENSORS
embedded screen at (239,245)-(555,339): ZLIB_VALVE_1_SENSORS
embedded screen at (239,554)-(561,593): VDIGIN
embedded screen at (239,340)-(554,375): VDIGIN
embedded screen at (239,515)-(555,552): VDIGIN
embedded screen at (239,597)-(557,636): VDIGIN
embedded screen at (239,471)-(556,506): VDIGIN
embedded screen at (767,222)-(1021,635): ZLIB_7211_Achse
embedded screen at (646,161)-(701,643): ZUFUEHRUNG_206POL
rectangle at (244,119)-(415,140): text "206 polig"; invisible if TRUE
rectangle at (774,227)-(945,248): text "ST03_51_M1"; invisible if TRUE
embedded screen at (698,117)-(1011,152): VDIGOUT_SMAL
rectangle at (698,117)-(869,138): text "ST00_73_K3"; invisible if TRUE
*)

(* Visualisation 01_ManualMode/ST03/MANUAL_ST03_7
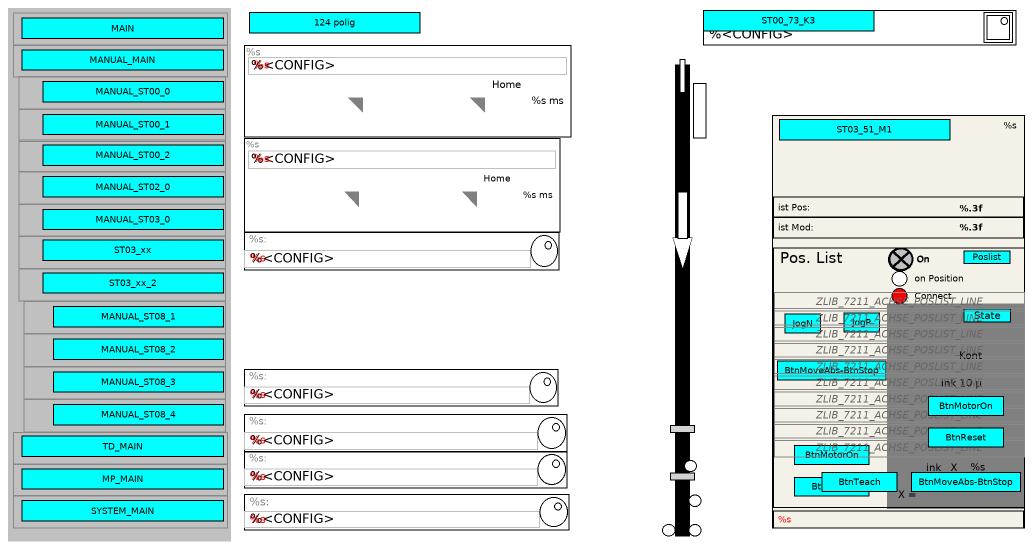
embedded screen at (3,115)-(226,648): M0000_Manual
embedded screen at (239,152)-(566,244): ZLIB_VALVE_1_SENSORS
embedded screen at (239,245)-(555,339): ZLIB_VALVE_1_SENSORS
embedded screen at (239,558)-(562,595): VDIGIN
embedded screen at (239,339)-(554,377): VDIGIN
embedded screen at (239,521)-(562,559): VDIGIN
embedded screen at (239,601)-(564,637): VDIGIN
embedded screen at (239,476)-(553,513): VDIGIN
embedded screen at (767,222)-(1021,635): ZLIB_7211_Achse
embedded screen at (646,161)-(701,643): ZUFUEHRUNG_124POL
rectangle at (244,119)-(415,140): text "124 polig"; invisible if TRUE
rectangle at (774,226)-(945,247): text "ST03_51_M1"; invisible if TRUE
embedded screen at (698,117)-(1011,152): VDIGOUT_SMAL
rectangle at (698,117)-(869,138): text "ST00_73_K3"; invisible if TRUE
*)

(* Visualisation 01_ManualMode/ST03/MANUAL_ST03_8
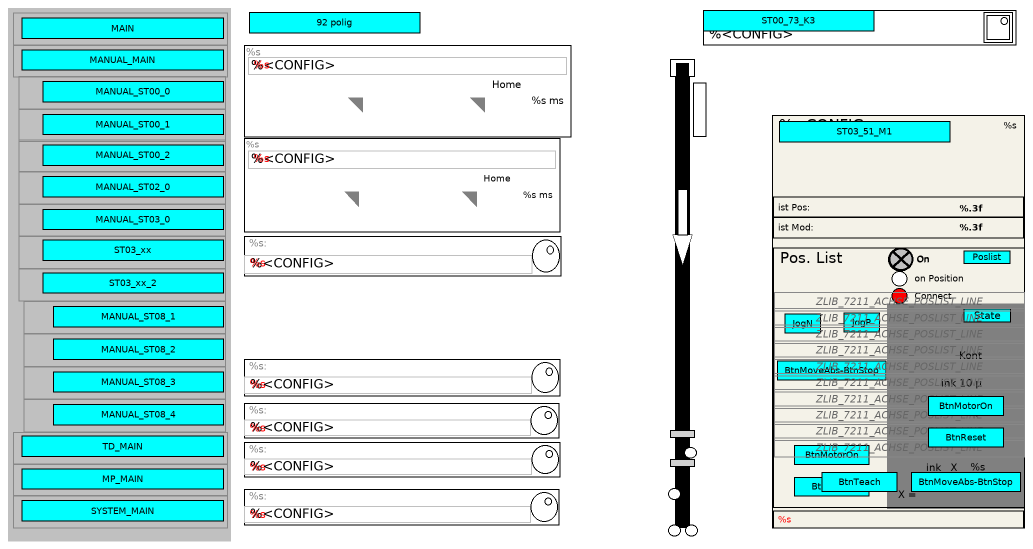
embedded screen at (3,115)-(226,648): M0000_Manual
embedded screen at (239,152)-(566,244): ZLIB_VALVE_1_SENSORS
embedded screen at (239,245)-(555,339): ZLIB_VALVE_1_SENSORS
embedded screen at (239,549)-(555,584): VDIGIN
embedded screen at (239,343)-(556,383): VDIGIN
embedded screen at (239,510)-(554,545): VDIGIN
embedded screen at (239,596)-(554,632): VDIGIN
embedded screen at (239,466)-(555,503): VDIGIN
embedded screen at (767,222)-(1021,635): ZLIB_7211_Achse
embedded screen at (646,161)-(701,643): ZUFUEHRUNG_92POL
rectangle at (244,119)-(415,140): text "92 polig"; invisible if TRUE
rectangle at (774,228)-(945,249): text "ST03_51_M1"; invisible if TRUE
embedded screen at (698,117)-(1011,152): VDIGOUT_SMAL
rectangle at (698,117)-(869,138): text "ST00_73_K3"; invisible if TRUE
*)

(* Visualisation 01_ManualMode/ST03/MANUAL_ST03_9
